{attribute 'qualified_only'}
{attribute 'to_string'}
TYPE eTcaWorkpieceStatus :
(
	undefined := 0, //leer
	noProcessDone, // grau
	laserProcessDone, // blau
	bondingAgentProcessDone, // orange
	castingProcessDone, //  violett
	finishProcessDone, //grün
	

	MAXSIZE
);
END_TYPE

(* stored: Version 1.1.0.1
   DUT eTcaWorkpieceStatus: Id {d29c626f-62d9-4d08-87c8-1233417dc64f} *)
